FUNCTION_BLOCK ServoNC EXTENDS FBA_Drive IMPLEMENTS I_EncodedDrive
VAR_OUTPUT	
	ready : BOOL;
	position : LREAL;
	velocity : LREAL;
END_VAR
VAR
	axis : AXIS_REF;
	
	mcReadPosition : MC_ReadActualPosition;
	mcReadVelocity : MC_ReadActualVelocity;
	mcReadError : MC_ReadAxisError;
	mcReset : MC_Reset;
	
	mcPower : MC_Power;
	mcMoveAbsolute : MC_MoveAbsolute;
	mcMoveRelative : MC_MoveRelative;
	mcMoveVelocity : MC_MoveVelocity;
	
	mcSetPosition : MC_SetPosition;
	mcStop : MC_Stop;
END_VAR
VAR_STAT CONSTANT
	targetingVelocity : INT := 500;
	continuousVelocity : INT := 100;
END_VAR

override();

blocks();

mcReset.Execute := FALSE;
mcMoveAbsolute.Execute := FALSE;
mcMoveRelative.Execute := FALSE;
mcMoveVelocity.Execute := FALSE;
mcSetPosition.Execute := FALSE;
mcStop.Execute := FALSE;

blocks();

ready := bEnable AND NOT Active AND HomeSet;

PROPERTY Active : BOOL
GET
Active := 
	mcMoveAbsolute.Busy OR 
	mcMoveRelative.Busy OR 
	mcMoveVelocity.Busy OR 
	mcSetPosition.Busy OR 
	mcReset.Busy OR 
	mcStop.Busy OR 
	step <> 0;
END_GET
END_PROPERTY

METHOD PRIVATE blocks : BOOL
mcReadPosition(
	Axis:= axis, 
	Enable:= TRUE, 
	Valid=> , 
	Busy=> , 
	Error=> , 
	ErrorID=> , 
	Position=> position);
	
mcReadVelocity(
	Axis:= axis, 
	Enable:= TRUE, 
	Valid=> , 
	Busy=> , 
	Error=> , 
	ErrorID=> , 
	ActualVelocity=> velocity);
	
mcReadError(
	Axis:= axis, 
	Enable:= TRUE, 
	Valid=> , 
	Busy=> , 
	Error=> , 
	ErrorID=> , 
	AxisErrorID=> );

mcReset(
	Axis:= axis, 
	Execute:= , 
	Done=> , 
	Busy=> , 
	Error=> , 
	ErrorID=> );

mcPower(
	Axis:= axis, 
	Enable:= bEnable, 
	Enable_Positive:= TRUE, 
	Enable_Negative:= TRUE, 
	Override:= 100, 
	BufferMode:= , 
	Options:= , 
	Status=> , 
	Busy=> , 
	Active=> , 
	Error=> , 
	ErrorID=> );

mcMoveAbsolute(
	Axis:= axis, 
	Execute:= , 
	Position:= , 
	Velocity:= targetingVelocity, 
	Acceleration:= , 
	Deceleration:= , 
	Jerk:= , 
	BufferMode:= , 
	Options:= , 
	Done=> , 
	Busy=> , 
	Active=> , 
	CommandAborted=> , 
	Error=> , 
	ErrorID=> );
	
mcMoveRelative(
	Axis:= axis, 
	Execute:= , 
	Distance:= ,
	Velocity:= targetingVelocity, 
	Acceleration:= , 
	Deceleration:= , 
	Jerk:= , 
	BufferMode:= , 
	Options:= , 
	Done=> , 
	Busy=> , 
	Active=> , 
	CommandAborted=> , 
	Error=> , 
	ErrorID=> );
	
mcMoveVelocity( //stopped with stop();
	Axis:= axis, 
	Execute:= , 
	Velocity:= continuousVelocity, 
	Acceleration:= , 
	Deceleration:= , 
	Jerk:= , 
	Direction:= , 
	BufferMode:= , 
	Options:= , 
	InVelocity=> , 
	Busy=> , 
	Active=> , 
	CommandAborted=> , 
	Error=> , 
	ErrorID=> );
	
mcSetPosition(
	Axis:= axis, 
	Execute:= , 
	Position:= , 
	Mode:= , 
	Options:= , 
	Done=> , 
	Busy=> , 
	Error=> , 
	ErrorID=> );
	
mcStop(
	Axis:= axis, 
	Execute:= , 
	Deceleration:= , 
	Jerk:= , 
	Options:= , 
	Done=> , 
	Busy=> , 
	Active=> , 
	CommandAborted=> , 
	Error=> , 
	ErrorID=> );
END_METHOD

PROPERTY CurrentPosition : LREAL
GET
CurrentPosition := position;
END_GET
SET
position := CurrentPosition;
END_SET
END_PROPERTY

PROPERTY Error : BOOL
GET
error := 
	mcMoveAbsolute.Error OR 
	mcMoveRelative.Error OR 
	mcMoveVelocity.Error OR 
	mcSetPosition.Error OR 
	mcReset.Error OR 
	mcStop.Error OR
	mcReadError.AxisErrorID > 0;
END_GET
END_PROPERTY

METHOD homingSequence : BOOL
CASE step OF
	Homing.IDLE:
		reset();
		IF bEnable THEN
			step := Homing.START;
		END_IF
		
	Homing.START:
		IF AtHome THEN
			mcMoveVelocity.Execute := FALSE;
			step := Homing.STOP;
			
		ELSIF AtInnerLimit THEN
			mcMoveVelocity.Execute := FALSE;
			step := Homing.RETRY;
			
		ELSE
			mcMoveVelocity.Direction := MC_Negative_Direction;
			mcMoveVelocity.Execute := NOT mcMoveVelocity.Execute;
		END_IF
		
	Homing.RETRY:
		IF AtOuterLimit THEN
			mcMoveVelocity.Execute := FALSE;
			step := Homing.START;
		ELSE
			mcMoveVelocity.Direction := MC_Positive_Direction;
			mcMoveVelocity.Execute := NOT mcMoveVelocity.Execute;
		END_IF
		
	Homing.STOP:
		IF velocity = 0 THEN
			mcStop.Execute := FALSE;
			step := Homing.SET;
		ELSE
			mcStop.Execute := TRUE;
		END_IF
		
	Homing.SET:
		IF position = 0 THEN
			mcSetPosition.Execute := FALSE;
			homingSequence := TRUE;
			step := Homing.DONE;
		ELSE
			mcSetPosition.Position := 0;
			mcSetPosition.Execute := TRUE;
		END_IF
		
	Homing.DONE:
		homingComplete := TRUE;
		step := Homing.IDLE;
		
END_CASE
END_METHOD

METHOD moveAbsolute : BOOL
VAR_INPUT
	newTarget : LREAL;
END_VAR
(*
VAR_OUTPUT
	fault : BOOL;
END_VAR
*)
IF NOT Active AND NOT error THEN
	mcMoveAbsolute.Position := newTarget;
	mcMoveAbsolute.Execute := TRUE;
END_IF

moveAbsolute := (*mcMoveAbsolute.Done AND mcMoveAbsolute.Active;*)
	position = newTarget;
END_METHOD

METHOD moveContinuous : BOOL
VAR_INPUT
	//direction : BOOL; //direction (F = inwards, T = outwards)
	direction : MC_Direction;
END_VAR
(*
IF mcMoveVelocity.Active THEN
	stop();
END_IF

IF NOT mcStop.Done THEN
	RETURN;
END_IF
*)
(*
IF direction THEN
	mcMoveVelocity.Direction := MC_Positive_Direction;
ELSE
	mcMoveVelocity.Direction := MC_Negative_Direction;
END_IF
*)
mcMoveVelocity.Direction := direction;

IF NOT mcMoveVelocity.Error THEN
	mcMoveVelocity.Execute := TRUE;
	moveContinuous := TRUE;
END_IF
END_METHOD

METHOD moveRelative : BOOL
VAR_INPUT
	distance : LREAL;
END_VAR
mcMoveRelative.Distance := distance;

moveRelative := mcMoveRelative.Done;
END_METHOD

METHOD PRIVATE override : BOOL
VAR_INPUT
END_VAR
(*
-at home and attempting to traverse outward
-at outer limit and attempting to traverse outward
-at inner limit and attempting to traverse inwards
*)
(*
inward = negative direction, negative velocity
outward = positive direction, positive velocity
*)

IF error THEN
	stop();
	reset();
	
ELSIF
	AtHome AND (TargetPosition > CurrentPosition OR velocity > 0) OR
	AtInnerLimit AND (TargetPosition > CurrentPosition OR velocity > 0) OR
	AtOuterLimit AND (TargetPosition < CurrentPosition OR velocity < 0)
THEN
	stop();
END_IF
END_METHOD

METHOD reset : BOOL
VAR_INPUT
END_VAR
mcReset.Execute := TRUE;

reset := mcReset.Done;
END_METHOD

METHOD stop : BOOL
VAR_INPUT
END_VAR
mcStop.Execute := TRUE;

mcMoveAbsolute.Execute := FALSE;
mcMoveRelative.Execute := FALSE;
mcMoveVelocity.Execute := FALSE;
END_METHOD

PROPERTY TargetPosition : LREAL
GET
END_GET
SET
moveAbsolute(newTarget := TargetPosition);
END_SET
END_PROPERTY

METHOD toHome : BOOL
VAR_INPUT
END_VAR
moveAbsolute(newTarget := 0);

toHome := AtHome;
END_METHOD

END_FUNCTION_BLOCK

(* stored: Version 1.1.0.1, ProductVersion 3.1.4024.11
   POU ServoNC: Id {bb489ff1-3ac2-4df2-9f8e-6593599f4fee}, SpecialFunc None
   Folder Private: Id {94f08eac-dbd6-4a1e-bdcc-cb414a065eb4}
   Folder Properties: Id {29bdcbf7-b9bd-446d-8be5-d556a3842a49}
   Property Active: Id {56a2da6d-8d1b-4f83-92b2-9ea1f87c2d8e}
   Get Get: Id {f234ae15-8868-413a-bfce-6f48ea7cc378}
   Method blocks: Id {4f63cb06-7dcb-4edd-943f-7b4c1e739caa}
   Property CurrentPosition: Id {543db0b5-6340-4956-a560-303a0c9d858d}
   Get Get: Id {961ec8ce-d029-49e4-afed-a15fd3c4099a}
   Set Set: Id {7790d45a-a505-4db9-b57a-0f249d291eda}
   Property Error: Id {4442e834-c433-49b0-80b7-e71b4f882d8e}
   Get Get: Id {4f349302-2e58-4461-b38f-ba1f4f81301c}
   Method homingSequence: Id {f083fc12-10be-475b-b5ad-e0e54c600219}
   Method moveAbsolute: Id {98b6f5bc-d22b-4bd2-89f6-c4bb4f9735b3}
   Method moveContinuous: Id {af66a590-1991-49ac-a629-d3f855ed14a2}
   Method moveRelative: Id {aea46495-93af-47b8-9cbc-949106d2ff4b}
   Method override: Id {9198b082-7fc7-4784-89da-f40da24b33ce}
   Method reset: Id {6ffa5af9-c14c-41dc-b194-ebef8b377ecd}
   Method stop: Id {4dccf70c-31b8-4d3e-a0e2-7db314723f88}
   Property TargetPosition: Id {b7fb16bd-29bf-4c77-ae2f-26ec2a5a948a}
   Get Get: Id {79e8370a-38ac-4b91-b49f-4b3721461425}
   Set Set: Id {3a85e76a-1c49-481e-8f9a-ba154f52f482}
   Method toHome: Id {863f6818-a649-4d05-aa71-7f25c03f5145} *)
